{attribute 'qualified_only'}
VAR_GLOBAL
	//cycle times
	tTaskCycleTime_MAIN				: TIME := T#50MS;
	tCtrlCycleTime_MAIN				: TIME := T#5S;
	
	//ip addresses
	sIP_EMAG_GT	: STRING := 'opc.tcp://192.168.116.33:4840';
	sIP_FlywheelMassStorage : STRING := 'opc.tcp://192.168.116.110:4840';
	sIP_MAFAC_Java : STRING := 'opc.tcp://192.168.116.47:4840';
	sIP_BvL_CleaningSystem : STRING := 'opc.tcp://192.168.116.129:4840';
	sIP_Annealing_Oven : STRING := 'opc.tcp://192.168.116.16:4840';
	sIP_DC : STRING := 'opc.tcp://192.168.116.41:4840';
	sIP_AbsorptionChiller : STRING := 'opc.tcp://192.168.116.56:4840'; 
	sIP_ImmersionHeater		: STRING := 'opc.tcp://192.168.115.56:4840';
	sIP_HES		: STRING := 'opc.tcp://192.168.115.71:4840';	
	sIP_CompressionChiller		: STRING := 'opc.tcp://192.168.116.19:4840';
	sIP_EMAG_VLC100	: STRING := 'opc.tcp://192.168.116.24:4840';
	sIP_HydraulicDemonstrator : STRING := 'opc.tcp://192.168.115.176:4840';
	sIP_Ventilation : STRING := '192.168.116.58';
	sIP_CHP1 : STRING := '192.168.116.118';
	sIP_CHP2 : STRING := '192.168.116.119';
	sIP_Emonio_HNHT_HeatPump : STRING := '192.168.116.173';
	sIP_Emonio_CN_HeatPump : STRING := '192.168.116.174';
	sIP_Emonio_eChiller : STRING := '192.168.116.177';
	sIP_Emonio_CondensingBoiler : STRING := '192.168.116.179';
END_VAR

(* stored: Version 1.1.0.1, ProductVersion 3.1.4024.10
   GVL GlobalVariables: Id {03b0febb-bd51-42dd-a1dc-b1b77f4022cb} *)
